PROGRAM POU
VAR
END_VAR

// NETWORK 1

END_PROGRAM

(* stored: Version 1.1.0.1, ProductVersion 3.1.4024.12
   POU POU: Id {129169f4-f6fd-4abc-8ea5-712222692328}, SpecialFunc None *)
